(* CODESYS project ai_oven_00_90.project
   Description: Receives some incoming messages and echoes them with CAN-ID +1
   Author: 3S - Smart Software Solutions GmbH
   Version: 1.0.0.0
   Title: CAN Bus API Example
   Company: 3S - Smart Software Solutions GmbH

Project tree, tasks and I/O mapping:
  xLH : CODESYS Control for Raspberry Pi 64 SL, CODESYS, order no. 2302000009, version 4.18.0.0
    application app
      libraries: Standard, 3.5.18.0 (System); Memory, * (3S - Smart Software Solutions GmbH); Util, 3.5.21.0 (System); VisuDialogs, * (System); CAA Tick Extern, 3.5.17.0 (CAA Technical Workgroup); SysTime, 3.5.17.0 (System); CmpIecTask, * (System); StringUtils, 3.5.20.0 (System); MQTT Client SL, 1.12.0.0 (CODESYS)
      task MAIN_TASK (cyclic, interval 20 ms, priority 0) calls MAIN
      task VISU_TASK (cyclic, interval 100 ms, priority 31) calls VisuElems.Visu_Prg
      visualisation Visualization
      program MAIN [ST]
      Symbols
      function block FB_PT1 [ST]: reset
    SoftMotion General Axis Pool
    GPIOs_A_B : GPIOs B+/Pi2, CODESYS, version 4.18.0.0
        unmapped channels: digital inputs (GPIO0..GPIO31), digital outputs (GPIO0..GPIO31)
    Onewire
    Camera device
      <Leer>
    SPI
    I²C
  libraries: VisuSymbols, 4.5.0.0 (System); DepictorBase, 1.2.0.0 (CODESYS)
  text list GlobalTextList
*)

// xLH/app/MAIN
PROGRAM MAIN
VAR
	fOvenTemperatureSetpoint: LREAL := 180.0;
	fOvenTemperature: LREAL;
	bOven: BOOL := TRUE;
	fbPt1Oven: FB_PT1 := (fK:=1.0, fT:=10.0);
END_VAR

IF bOven THEN
	fbPt1Oven.fX := fOvenTemperatureSetpoint; 
ELSE
	fbPt1Oven.fX := 20.0;
END_IF
fbPt1Oven();
fOvenTemperature := fbPt1Oven.fY;

END_PROGRAM

// xLH/app/FB_PT1
{attribute 'FBVisuCreator'}
{attribute 'FBVisuCreatorPrefix' :=  'RET_VISU_'}
FUNCTION_BLOCK FB_PT1
VAR_INPUT
	fX: LREAL;
	fK: LREAL;
	fT: LREAL;
	bReset: BOOL;
	fDt: LREAL := 0.020;
END_VAR
VAR_OUTPUT
	fY: LREAL;
END_VAR
VAR
	rSumme: LREAL;
END_VAR

IF bReset THEN
	reset();
END_IF

IF (fT > 0.0) THEN
	fY := fY + (-fY + fK*fX)/MAX(fT,0.001)*fDt;
ELSE
	fY := fX;
END_IF

ACTION reset:
fY := 0.0;
END_ACTION

END_FUNCTION_BLOCK

// xLH/app/Visualization
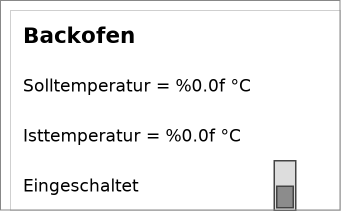
VISUALIZATION Visualization  // 341x211
    Rectangle (10,10 331x201)
    Rectangle (20,10 301x51), "Backofen"
    Rectangle (20,60 311x51), "Solltemperatur = %0.0f °C", text variable: MAIN.fOvenTemperatureSetpoint
        OnMouseClick: write the text variable via Default, min 100.0, max 300.0
    Rectangle (20,110 311x51), "Isttemperatur = %0.0f °C", text variable: MAIN.fOvenTemperature
    Rectangle (20,160 211x51), "Eingeschaltet", text variable: MAIN.fOvenTemperatureSetpoint
    DipSwitch (240,160 90x51), variable: MAIN.bOven, behaviour: TOGGLE, style: Switch-DipSwitch-Gray
END_VISUALIZATION
